// TIA Portal V20 export
// export: Created 2026-07-10T11:12:33.1539686Z, ExportSetting WithDefaults, DisplayName Totally Integrated Automation Portal, DisplayVersion V20, DisplayName TIA Portal Openness, DisplayVersion V20, DisplayName TIA Portal Version Control Interface, DisplayVersion V20, DisplayName STEP 7 Professional, DisplayVersion V20, DisplayName STEP 7 Safety, DisplayVersion V20, DisplayName WinCC Basic/Comfort/Advanced, DisplayVersion V20, DisplayName WinCC Unified, DisplayVersion V20
FUNCTION_BLOCK "MotorPositionNoFeedback"   // FB11, SCL
{ S7_Optimized_Access := 'TRUE' }
VERSION : 0.1
// stored: AutoNumber true, IsIECCheckEnabled false, IsRetainMemResEnabled false, MemoryReserve 100, SetENOAutomatically false, UDAEnableTagReadback false
   VAR_INPUT
      Enable : Bool;
      LimitSwitch0 : Bool;
      LimitSwitch100 : Bool;
      Invalidate : Bool := False;
      FullMovingTime : Real;
      LappingZone : Real := 1.0;
      Open : Bool;
      Close : Bool;
      SwitchAutoMode : Bool;
   END_VAR
   VAR_OUTPUT
      CurrentPosition : Real;
      Error : Bool := FALSE;
   END_VAR
   VAR
      PreviousPosition : Real;
      OnePercentImpulse : Real;
      MovingTimer1 { S7_SetPoint := 'True'} : TON_TIME;
      MovingTimer2 { S7_SetPoint := 'True'} : TON_TIME;
   END_VAR
BEGIN
   #LappingZone := LIMIT(MN := 1.0, IN := #LappingZone, MX := 30.0);

   IF #Enable THEN
       #MovingTimer1(IN:=#Open, PT:= DINT_TO_TIME(REAL_TO_DINT(#FullMovingTime)*1000/100));
       #MovingTimer2(IN:=#Close,PT:= DINT_TO_TIME(REAL_TO_DINT(#FullMovingTime)*1000/100));

       IF #Error = FALSE THEN
           IF #Open AND #MovingTimer1.Q THEN
               #CurrentPosition := #PreviousPosition + 1;
               #CurrentPosition := MIN(IN1 := #CurrentPosition, IN2 := 100-#LappingZone);
               RESET_TIMER(#MovingTimer1);
               #PreviousPosition := #CurrentPosition;
           END_IF;

           IF #Close AND #MovingTimer2.Q THEN
               #CurrentPosition := #PreviousPosition - 1;
               #CurrentPosition := MAX(IN1 := #CurrentPosition, IN2 := #LappingZone);
               RESET_TIMER(#MovingTimer2);
               #PreviousPosition := #CurrentPosition;
           END_IF;
       END_IF;

       IF #LimitSwitch100 THEN
           #CurrentPosition := 100;
           #Error := 0;
           #PreviousPosition := #CurrentPosition;
           RESET_TIMER(#MovingTimer1);
           RESET_TIMER(#MovingTimer2);
       END_IF;

       IF #LimitSwitch0 THEN
           #CurrentPosition := 0;
           #Error := 0;
           #PreviousPosition := #CurrentPosition;
           RESET_TIMER(#MovingTimer1);
           RESET_TIMER(#MovingTimer2);
       END_IF;

       IF #Invalidate THEN
           #CurrentPosition := 0;
           #Error := TRUE;
       END_IF;
   ELSE
       #CurrentPosition := 0;
       #Error := TRUE;
       RESET_TIMER(#MovingTimer1);
       RESET_TIMER(#MovingTimer2);
   END_IF;
END_FUNCTION_BLOCK
